 X = -308.2 mm, Y = 326.9 mm, Z = 531.8 mm,       W = -6.7 deg, P = 19.4 deg,
    GP2:
        UF : 1, UT : 2,
       J1 = 0.0 deg, J2 = 0.0 deg
 };
P[134] {
    GP1:
        UF : 6, UT : 5,     CONFIG: 'N U T, 0, 0, 0',
       X = -327.0 mm, Y = 261.3 mm, Z = 531.8 mm,
       W = -6.7 deg, P = 19.5 deg,
    GP2:
        UF : 1, UT : 2,
       J1 = 0.0 deg, J2 = 0.0 deg
 };
P[404] {
    GP1:
        UF : 6, UT : 5,     CONFIG: 'N U T, 0, 0, 0',
 X = -310.0 mm, Y = 332.3 mm, Z = 531.8 mm,       W = -6.7 deg, P = 19.5 deg,
    GP2:
        UF : 1, UT : 2,
       J1 = 0.0 deg, J2 = 0.0 deg
 };
P[135] {
    GP1:
        UF : 6, UT : 5,     CONFIG: 'N U T, 0, 0, 0',
       X = -328.0 mm, Y = 264.4 mm, Z = 531.8 mm,
       W = -7.3 deg, P = 19.2 deg,
    GP2:
        UF : 1, UT : 2,
       J1 = 0.0 deg, J2 = 0.0 deg
 };
P[405] {
    GP1:
        UF : 6, UT : 5,     CONFIG: 'N U T, 0, 0, 0',
 X = -311.0 mm, Y = 335.4 mm, Z = 531.8 mm,       W = -7.3 deg, P = 19.2 deg,
    GP2:
        UF : 1, UT : 2,
       J1 = 0.0 deg, J2 = 0.0 deg
 };
P[136] {
    GP1:
        UF : 6, UT : 5,     CONFIG: 'N U T, 0, 0, 0',
       X = -329.2 mm, Y = 267.4 mm, Z = 531.8 mm,
       W = -7.3 deg, P = 19.0 deg,
    GP2:
        UF : 1, UT : 2,
       J1 = 0.0 deg, J2 = 0.0 deg
 };
P[406] {
    GP1:
        UF : 6, UT : 5,     CONFIG: 'N U T, 0, 0, 0',
 X = -312.2 mm, Y = 338.4 mm, Z = 531.8 mm,       W = -7.3 deg, P = 19.0 deg,
    GP2:
        UF : 1, UT : 2,
       J1 = 0.0 deg, J2 = 0.0 deg
 };
P[137] {
    GP1:
        UF : 6, UT : 5,     CONFIG: 'N U T, 0, 0, 0',
       X = -330.4 mm, Y = 270.7 mm, Z = 531.8 mm,
       W = -7.2 deg, P = 18.9 deg,
    GP2:
        UF : 1, UT : 2,
       J1 = 0.0 deg, J2 = 0.0 deg
 };
P[407] {
    GP1:
        UF : 6, UT : 5,     CONFIG: 'N U T, 0, 0, 0',
 X = -313.4 mm, Y = 341.7 mm, Z = 531.8 mm,       W = -7.2 deg, P = 18.9 deg,
    GP2:
        UF : 1, UT : 2,
       J1 = 0.0 deg, J2 = 0.0 deg
 };
P[138] {
    GP1:
        UF : 6, UT : 5,     CONFIG: 'N U T, 0, 0, 0',
       X = -331.6 mm, Y = 273.8 mm, Z = 531.8 mm,
       W = -7.7 deg, P = 18.5 deg,
    GP2:
        UF : 1, UT : 2,
       J1 = 0.0 deg, J2 = 0.0 deg
 };
P[408] {
    GP1:
        UF : 6, UT : 5,     CONFIG: 'N U T, 0, 0, 0',
 X = -314.6 mm, Y = 344.8 mm, Z = 531.8 mm,       W = -7.7 deg, P = 18.5 deg,
    GP2:
        UF : 1, UT : 2,
       J1 = 0.0 deg, J2 = 0.0 deg
 };
P[139] {
    GP1:
        UF : 6, UT : 5,     CONFIG: 'N U T, 0, 0, 0',
       X = -332.8 mm, Y = 276.8 mm, Z = 531.8 mm,
       W = -7.7 deg, P = 18.5 deg,
    GP2:
        UF : 1, UT : 2,
       J1 = 0.0 deg, J2 = 0.0 deg
 };
P[409] {
    GP1:
        UF : 6, UT : 5,     CONFIG: 'N U T, 0, 0, 0',
 X = -315.8 mm, Y = 347.8 mm, Z = 531.8 mm,       W = -7.7 deg, P = 18.5 deg,
    GP2:
        UF : 1, UT : 2,
       J1 = 0.0 deg, J2 = 0.0 deg
 };
P[140] {
    GP1:
        UF : 6, UT : 5,     CONFIG: 'N U T, 0, 0, 0',
       X = -334.1 mm, Y = 280.0 mm, Z = 531.8 mm,
       W = -7.7 deg, P = 18.4 deg,
    GP2:
        UF : 1, UT : 2,
       J1 = 0.0 deg, J2 = 0.0 deg
 };
P[410] {
    GP1:
        UF : 6, UT : 5,     CONFIG: 'N U T, 0, 0, 0',
 X = -317.1 mm, Y = 351.0 mm, Z = 531.8 mm,       W = -7.7 deg, P = 18.4 deg,
    GP2:
        UF : 1, UT : 2,
       J1 = 0.0 deg, J2 = 0.0 deg
 };
P[141] {
    GP1:
        UF : 6, UT : 5,     CONFIG: 'N U T, 0, 0, 0',
       X = -335.3 mm, Y = 282.9 mm, Z = 531.8 mm,
       W = -8.2 deg, P = 18.1 deg,
    GP2:
        UF : 1, UT : 2,
       J1 = 0.0 deg, J2 = 0.0 deg
 };
P[411] {
    GP1:
        UF : 6, UT : 5,     CONFIG: 'N U T, 0, 0, 0',
 X = -318.3 mm, Y = 353.9 mm, Z = 531.8 mm,       W = -8.2 deg, P = 18.1 deg,
    GP2:
        UF : 1, UT : 2,
       J1 = 0.0 deg, J2 = 0.0 deg
 };
P[142] {
    GP1:
        UF : 6, UT : 5,     CONFIG: 'N U T, 0, 0, 0',
       X = -336.6 mm, Y = 285.8 mm, Z = 531.8 mm,
       W = -8.2 deg, P = 18.0 deg,
    GP2:
        UF : 1, UT : 2,
       J1 = 0.0 deg, J2 = 0.0 deg
 };
P[412] {
    GP1:
        UF : 6, UT : 5,     CONFIG: 'N U T, 0, 0, 0',
 X = -319.6 mm, Y = 356.8 mm, Z = 531.8 mm,       W = -8.2 deg, P = 18.0 deg,
    GP2:
        UF : 1, UT : 2,
       J1 = 0.0 deg, J2 = 0.0 deg
 };
P[143] {
    GP1:
        UF : 6, UT : 5,     CONFIG: 'N U T, 0, 0, 0',
       X = -338.1 mm, Y = 289.2 mm, Z = 531.8 mm,
       W = -8.1 deg, P = 17.9 deg,
    GP2:
        UF : 1, UT : 2,
       J1 = 0.0 deg, J2 = 0.0 deg
 };
P[413] {
    GP1:
        UF : 6, UT : 5,     CONFIG: 'N U T, 0, 0, 0',
 X = -321.1 mm, Y = 360.2 mm, Z = 531.8 mm,       W = -8.1 deg, P = 17.9 deg,
    GP2:
        UF : 1, UT : 2,
       J1 = 0.0 deg, J2 = 0.0 deg
 };
P[144] {
    GP1:
        UF : 6, UT : 5,     CONFIG: 'N U T, 0, 0, 0',
       X = -339.3 mm, Y = 291.9 mm, Z = 531.8 mm,
       W = -8.7 deg, P = 17.5 deg,
    GP2:
        UF : 1, UT : 2,
       J1 = 0.0 deg, J2 = 0.0 deg
 };
P[414] {
    GP1:
        UF : 6, UT : 5,     CONFIG: 'N U T, 0, 0, 0',
 X = -322.3 mm, Y = 362.9 mm, Z = 531.8 mm,       W = -8.7 deg, P = 17.5 deg,
    GP2:
        UF : 1, UT : 2,
       J1 = 0.0 deg, J2 = 0.0 deg
 };
P[145] {
    GP1:
        UF : 6, UT : 5,     CONFIG: 'N U T, 0, 0, 0',
       X = -343.7 mm, Y = 300.7 mm, Z = 531.8 mm,
       W = -9.1 deg, P = 16.9 deg,
    GP2:
        UF : 1, UT : 2,
       J1 = 0.0 deg, J2 = 0.0 deg
 };
P[415] {
    GP1:
        UF : 6, UT : 5,     CONFIG: 'N U T, 0, 0, 0',
 X = -326.7 mm, Y = 371.7 mm, Z = 531.8 mm,       W = -9.1 deg, P = 16.9 deg,
    GP2:
        UF : 1, UT : 2,
       J1 = 0.0 deg, J2 = 0.0 deg
 };
P[146] {
    GP1:
        UF : 6, UT : 5,     CONFIG: 'N U T, 0, 0, 0',
       X = -345.2 mm, Y = 303.6 mm, Z = 531.8 mm,
       W = -9.1 deg, P = 16.8 deg,
    GP2:
        UF : 1, UT : 2,
       J1 = 0.0 deg, J2 = 0.0 deg
 };
P[416] {
    GP1:
        UF : 6, UT : 5,     CONFIG: 'N U T, 0, 0, 0',
 X = -328.2 mm, Y = 374.6 mm, Z = 531.8 mm,       W = -9.1 deg, P = 16.8 deg,
    GP2:
        UF : 1, UT : 2,
       J1 = 0.0 deg, J2 = 0.0 deg
 };
P[147] {
    GP1:
        UF : 6, UT : 5,     CONFIG: 'N U T, 0, 0, 0',
       X = -347.1 mm, Y = 307.0 mm, Z = 531.8 mm,
       W = -9.1 deg, P = 16.7 deg,
    GP2:
        UF : 1, UT : 2,
       J1 = 0.0 deg, J2 = 0.0 deg
 };
P[417] {
    GP1:
        UF : 6, UT : 5,     CONFIG: 'N U T, 0, 0, 0',
 X = -330.1 mm, Y = 378.0 mm, Z = 531.8 mm,       W = -9.1 deg, P = 16.7 deg,
    GP2:
        UF : 1, UT : 2,
       J1 = 0.0 deg, J2 = 0.0 deg
 };
P[148] {
    GP1:
        UF : 6, UT : 5,     CONFIG: 'N U T, 0, 0, 0',
       X = -348.5 mm, Y = 309.7 mm, Z = 531.8 mm,
       W = -9.5 deg, P = 16.4 deg,
    GP2:
        UF : 1, UT : 2,
       J1 = 0.0 deg, J2 = 0.0 deg
 };
P[418] {
    GP1:
        UF : 6, UT : 5,     CONFIG: 'N U T, 0, 0, 0',
 X = -331.5 mm, Y = 380.7 mm, Z = 531.8 mm,       W = -9.5 deg, P = 16.4 deg,
    GP2:
        UF : 1, UT : 2,
       J1 = 0.0 deg, J2 = 0.0 deg
 };
P[149] {
    GP1:
        UF : 6, UT : 5,     CONFIG: 'N U T, 0, 0, 0',
       X = -353.5 mm, Y = 318.3 mm, Z = 531.8 mm,
       W = -9.9 deg, P = 15.9 deg,
    GP2:
        UF : 1, UT : 2,
       J1 = 0.0 deg, J2 = 0.0 deg
 };
P[419] {
    GP1:
        UF : 6, UT : 5,     CONFIG: 'N U T, 0, 0, 0',
 X = -336.5 mm, Y = 389.3 mm, Z = 531.8 mm,       W = -9.9 deg, P = 15.9 deg,
    GP2:
        UF : 1, UT : 2,
       J1 = 0.0 deg, J2 = 0.0 deg
 };
P[150] {
    GP1:
        UF : 6, UT : 5,     CONFIG: 'N U T, 0, 0, 0',
       X = -358.7 mm, Y = 326.6 mm, Z = 531.8 mm,
       W = -10.1 deg, P = 15.4 deg,
    GP2:
        UF : 1, UT : 2,
       J1 = 0.0 deg, J2 = 0.0 deg
 };
P[420] {
    GP1:
        UF : 6, UT : 5,     CONFIG: 'N U T, 0, 0, 0',
 X = -341.7 mm, Y = 397.6 mm, Z = 531.8 mm,       W = -10.1 deg, P = 15.4 deg,
    GP2:
        UF : 1, UT : 2,
       J1 = 0.0 deg, J2 = 0.0 deg
 };
P[151] {
    GP1:
        UF : 6, UT : 5,     CONFIG: 'N U T, 0, 0, 0',
       X = -364.2 mm, Y = 334.9 mm, Z = 531.8 mm,
       W = -10.4 deg, P = 14.9 deg,
    GP2:
        UF : 1, UT : 2,
       J1 = 0.0 deg, J2 = 0.0 deg
 };
P[421] {
    GP1:
        UF : 6, UT : 5,     CONFIG: 'N U T, 0, 0, 0',
 X = -347.2 mm, Y = 405.9 mm, Z = 531.8 mm,       W = -10.4 deg, P = 14.9 deg,
    GP2:
        UF : 1, UT : 2,
       J1 = 0.0 deg, J2 = 0.0 deg
 };
P[152] {
    GP1:
        UF : 6, UT : 5,     CONFIG: 'N U T, 0, 0, 0',
       X = -369.8 mm, Y = 342.9 mm, Z = 531.8 mm,
       W = -10.6 deg, P = 14.5 deg,
    GP2:
        UF : 1, UT : 2,
       J1 = 0.0 deg, J2 = 0.0 deg
 };
P[422] {
    GP1:
        UF : 6, UT : 5,     CONFIG: 'N U T, 0, 0, 0',
 X = -352.8 mm, Y = 413.9 mm, Z = 531.8 mm,       W = -10.6 deg, P = 14.5 deg,
    GP2:
        UF : 1, UT : 2,
       J1 = 0.0 deg, J2 = 0.0 deg
 };
P[153] {
    GP1:
        UF : 6, UT : 5,     CONFIG: 'N U T, 0, 0, 0',
       X = -375.7 mm, Y = 350.9 mm, Z = 531.8 mm,
       W = -11.0 deg, P = 14.1 deg,
    GP2:
        UF : 1, UT : 2,
       J1 = 0.0 deg, J2 = 0.0 deg
 };
P[423] {
    GP1:
        UF : 6, UT : 5,     CONFIG: 'N U T, 0, 0, 0',
 X = -358.7 mm, Y = 421.9 mm, Z = 531.8 mm,       W = -11.0 deg, P = 14.1 deg,
    GP2:
        UF : 1, UT : 2,
       J1 = 0.0 deg, J2 = 0.0 deg
 };
P[154] {
    GP1:
        UF : 6, UT : 5,     CONFIG: 'N U T, 0, 0, 0',
       X = -381.9 mm, Y = 358.6 mm, Z = 531.8 mm,
       W = -11.4 deg, P = 13.8 deg,
    GP2:
        UF : 1, UT : 2,
       J1 = 0.0 deg, J2 = 0.0 deg
 };
P[424] {
    GP1:
        UF : 6, UT : 5,     CONFIG: 'N U T, 0, 0, 0',
 X = -364.9 mm, Y = 429.6 mm, Z = 531.8 mm,       W = -11.4 deg, P = 13.8 deg,
    GP2:
        UF : 1, UT : 2,
       J1 = 0.0 deg, J2 = 0.0 deg
 };
P[155] {
    GP1:
        UF : 6, UT : 5,     CONFIG: 'N U T, 0, 0, 0',
       X = -388.2 mm, Y = 366.1 mm, Z = 531.8 mm,
       W = -11.5 deg, P = 13.2 deg,
    GP2:
        UF : 1, UT : 2,
       J1 = 0.0 deg, J2 = 0.0 deg
 };
P[425] {
    GP1:
        UF : 6, UT : 5,     CONFIG: 'N U T, 0, 0, 0',
 X = -371.2 mm, Y = 437.1 mm, Z = 531.8 mm,       W = -11.5 deg, P = 13.2 deg,
    GP2:
        UF : 1, UT : 2,
       J1 = 0.0 deg, J2 = 0.0 deg
 };
P[156] {
    GP1:
        UF : 6, UT : 5,     CONFIG: 'N U T, 0, 0, 0',
       X = -394.8 mm, Y = 373.5 mm, Z = 531.8 mm,
       W = -11.7 deg, P = 12.5 deg,
    GP2:
        UF : 1, UT : 2,
       J1 = 0.0 deg, J2 = 0.0 deg
 };
P[426] {
    GP1:
        UF : 6, UT : 5,     CONFIG: 'N U T, 0, 0, 0',
 X = -377.8 mm, Y = 444.5 mm, Z = 531.8 mm,       W = -11.7 deg, P = 12.5 deg,
    GP2:
        UF : 1, UT : 2,
       J1 = 0.0 deg, J2 = 0.0 deg
 };
P[157] {
    GP1:
        UF : 6, UT : 5,     CONFIG: 'N U T, 0, 0, 0',
       X = -401.6 mm, Y = 380.6 mm, Z = 531.8 mm,
       W = -11.8 deg, P = 12.0 deg,
    GP2:
        UF : 1, UT : 2,
       J1 = 0.0 deg, J2 = 0.0 deg
 };
P[427] {
    GP1:
        UF : 6, UT : 5,     CONFIG: 'N U T, 0, 0, 0',
 X = -384.6 mm, Y = 451.6 mm, Z = 531.8 mm,       W = -11.8 deg, P = 12.0 deg,
    GP2:
        UF : 1, UT : 2,
       J1 = 0.0 deg, J2 = 0.0 deg
 };
P[158] {
    GP1:
        UF : 6, UT : 5,     CONFIG: 'N U T, 0, 0, 0',
       X = -408.7 mm, Y = 387.5 mm, Z = 531.8 mm,
       W = -11.7 deg, P = 11.3 deg,
    GP2:
        UF : 1, UT : 2,
       J1 = 0.0 deg, J2 = 0.0 deg
 };
P[428] {
    GP1:
        UF : 6, UT : 5,     CONFIG: 'N U T, 0, 0, 0',
 X = -391.7 mm, Y = 458.5 mm, Z = 531.8 mm,       W = -11.7 deg, P = 11.3 deg,
    GP2:
        UF : 1, UT : 2,
       J1 = 0.0 deg, J2 = 0.0 deg
 };
P[159] {
    GP1:
        UF : 6, UT : 5,     CONFIG: 'N U T, 0, 0, 0',
       X = -415.9 mm, Y = 394.3 mm, Z = 531.8 mm,
       W = -11.7 deg, P = 10.7 deg,
    GP2:
        UF : 1, UT : 2,
       J1 = 0.0 deg, J2 = 0.0 deg
 };
P[429] {
    GP1:
        UF : 6, UT : 5,     CONFIG: 'N U T, 0, 0, 0',
 X = -398.9 mm, Y = 465.3 mm, Z = 531.8 mm,       W = -11.7 deg, P = 10.7 deg,
    GP2:
        UF : 1, UT : 2,
       J1 = 0.0 deg, J2 = 0.0 deg
 };
P[160] {
    GP1:
        UF : 6, UT : 5,     CONFIG: 'N U T, 0, 0, 0',
       X = -423.3 mm, Y = 400.8 mm, Z = 531.8 mm,
       W = -11.8 deg, P = 10.1 deg,
    GP2:
        UF : 1, UT : 2,
       J1 = 0.0 deg, J2 = 0.0 deg
 };
P[430] {
    GP1:
        UF : 6, UT : 5,     CONFIG: 'N U T, 0, 0, 0',
 X = -406.3 mm, Y = 471.8 mm, Z = 531.8 mm,       W = -11.8 deg, P = 10.1 deg,
    GP2:
        UF : 1, UT : 2,
       J1 = 0.0 deg, J2 = 0.0 deg
 };
P[161] {
    GP1:
        UF : 6, UT : 5,     CONFIG: 'N U T, 0, 0, 0',
       X = -425.5 mm, Y = 402.6 mm, Z = 531.8 mm,
       W = -11.9 deg, P = 9.9 deg,
    GP2:
        UF : 1, UT : 2,
       J1 = 0.0 deg, J2 = 0.0 deg
 };
P[431] {
    GP1:
        UF : 6, UT : 5,     CONFIG: 'N U T, 0, 0, 0',
 X = -408.5 mm, Y = 473.6 mm, Z = 531.8 mm,       W = -11.9 deg, P = 9.9 deg,
    GP2:
        UF : 1, UT : 2,
       J1 = 0.0 deg, J2 = 0.0 deg
 };
P[162] {
    GP1:
        UF : 6, UT : 5,     CONFIG: 'N U T, 0, 0, 0',
       X = -428.2 mm, Y = 404.9 mm, Z = 531.8 mm,
       W = -11.8 deg, P = 9.8 deg,
    GP2:
        UF : 1, UT : 2,
       J1 = 0.0 deg, J2 = 0.0 deg
 };
P[432] {
    GP1:
        UF : 6, UT : 5,     CONFIG: 'N U T, 0, 0, 0',
 X = -411.2 mm, Y = 475.9 mm, Z = 531.8 mm,       W = -11.8 deg, P = 9.8 deg,
    GP2:
        UF : 1, UT : 2,
       J1 = 0.0 deg, J2 = 0.0 deg
 };
P[163] {
    GP1:
        UF : 6, UT : 5,     CONFIG: 'N U T, 0, 0, 0',
       X = -429.4 mm, Y = 405.9 mm, Z = 531.8 mm,
       W = -11.5 deg, P = 10.1 deg,
    GP2:
        UF : 1, UT : 2,
       J1 = 0.0 deg, J2 = 0.0 deg
 };
P[433] {
    GP1:
        UF : 6, UT : 5,     CONFIG: 'N U T, 0, 0, 0',
 X = -412.4 mm, Y = 476.9 mm, Z = 531.8 mm,       W = -11.5 deg, P = 10.1 deg,
    GP2:
        UF : 1, UT : 2,
       J1 = 0.0 deg, J2 = 0.0 deg
 };
P[164] {
    GP1:
        UF : 6, UT : 5,     CONFIG: 'N U T, 0, 0, 0',
       X = -430.8 mm, Y = 407.1 mm, Z = 531.8 mm,
       W = -11.2 deg, P = 10.8 deg,
    GP2:
        UF : 1, UT : 2,
       J1 = 0.0 deg, J2 = 0.0 deg
 };
P[434] {
    GP1:
        UF : 6, UT : 5,     CONFIG: 'N U T, 0, 0, 0',
 X = -413.8 mm, Y = 478.1 mm, Z = 531.8 mm,       W = -11.2 deg, P = 10.8 deg,
    GP2:
        UF : 1, UT : 2,
       J1 = 0.0 deg, J2 = 0.0 deg
 };
P[165] {
    GP1:
        UF : 6, UT : 5,     CONFIG: 'N U T, 0, 0, 0',
       X = -431.4 mm, Y = 407.7 mm, Z = 531.8 mm,
       W = -11.0 deg, P = 11.1 deg,
    GP2:
        UF : 1, UT : 2,
       J1 = 0.0 deg, J2 = 0.0 deg
 };
P[435] {
    GP1:
        UF : 6, UT : 5,     CONFIG: 'N U T, 0, 0, 0',
 X = -414.4 mm, Y = 478.7 mm, Z = 531.8 mm,       W = -11.0 deg, P = 11.1 deg,
    GP2:
        UF : 1, UT : 2,
       J1 = 0.0 deg, J2 = 0.0 deg
 };
P[166] {
    GP1:
        UF : 6, UT : 5,     CONFIG: 'N U T, 0, 0, 0',
       X = -431.6 mm, Y = 407.9 mm, Z = 531.8 mm,
       W = -10.8 deg, P = 11.3 deg,
    GP2:
        UF : 1, UT : 2,
       J1 = 0.0 deg, J2 = 0.0 deg
 };
P[436] {
    GP1:
        UF : 6, UT : 5,     CONFIG: 'N U T, 0, 0, 0',
 X = -414.6 mm, Y = 478.9 mm, Z = 531.8 mm,       W = -10.8 deg, P = 11.3 deg,
    GP2:
        UF : 1, UT : 2,
       J1 = 0.0 deg, J2 = 0.0 deg
 };
P[167] {
    GP1:
        UF : 6, UT : 5,     CONFIG: 'N U T, 0, 0, 0',
       X = -431.7 mm, Y = 408.1 mm, Z = 531.8 mm,
       W = -10.6 deg, P = 11.6 deg,
    GP2:
        UF : 1, UT : 2,
       J1 = 0.0 deg, J2 = 0.0 deg
 };
P[437] {
    GP1:
        UF : 6, UT : 5,     CONFIG: 'N U T, 0, 0, 0',
 X = -414.7 mm, Y = 479.1 mm, Z = 531.8 mm,       W = -10.6 deg, P = 11.6 deg,
    GP2:
        UF : 1, UT : 2,
       J1 = 0.0 deg, J2 = 0.0 deg
 };
P[168] {
    GP1:
        UF : 6, UT : 5,     CONFIG: 'N U T, 0, 0, 0',
       X = -431.9 mm, Y = 408.2 mm, Z = 531.8 mm,
       W = -10.3 deg, P = 11.8 deg,
    GP2:
        UF : 1, UT : 2,
       J1 = 0.0 deg, J2 = 0.0 deg
 };
P[438] {
    GP1:
        UF : 6, UT : 5,     CONFIG: 'N U T, 0, 0, 0',
 X = -414.9 mm, Y = 479.2 mm, Z = 531.8 mm,       W = -10.3 deg, P = 11.8 deg,
    GP2:
        UF : 1, UT : 2,
       J1 = 0.0 deg, J2 = 0.0 deg
 };
P[169] {
    GP1:
        UF : 6, UT : 5,     CONFIG: 'N U T, 0, 0, 0',
       X = -432.0 mm, Y = 408.4 mm, Z = 531.8 mm,
       W = -10.1 deg, P = 12.1 deg,
    GP2:
        UF : 1, UT : 2,
       J1 = 0.0 deg, J2 = 0.0 deg
 };
P[439] {
    GP1:
        UF : 6, UT : 5,     CONFIG: 'N U T, 0, 0, 0',
 X = -415.0 mm, Y = 479.4 mm, Z = 531.8 mm,       W = -10.1 deg, P = 12.1 deg,
    GP2:
        UF : 1, UT : 2,
       J1 = 0.0 deg, J2 = 0.0 deg
 };
P[170] {
    GP1:
        UF : 6, UT : 5,     CONFIG: 'N U T, 0, 0, 0',
       X = -432.6 mm, Y = 409.1 mm, Z = 531.8 mm,
       W = -9.7 deg, P = 12.7 deg,
    GP2:
        UF : 1, UT : 2,
       J1 = 0.0 deg, J2 = 0.0 deg
 };
P[440] {
    GP1:
        UF : 6, UT : 5,     CONFIG: 'N U T, 0, 0, 0',
 X = -415.6 mm, Y = 480.1 mm, Z = 531.8 mm,       W = -9.7 deg, P = 12.7 deg,
    GP2:
        UF : 1, UT : 2,
       J1 = 0.0 deg, J2 = 0.0 deg
 };
P[171] {
    GP1:
        UF : 6, UT : 5,     CONFIG: 'N U T, 0, 0, 0',
       X = -433.2 mm, Y = 410.0 mm, Z = 531.8 mm,
       W = -9.5 deg, P = 12.9 deg,
    GP2:
        UF : 1, UT : 2,
       J1 = 0.0 deg, J2 = 0.0 deg
 };
P[441] {
    GP1:
        UF : 6, UT : 5,     CONFIG: 'N U T, 0, 0, 0',
 X = -416.2 mm, Y = 481.0 mm, Z = 531.8 mm,       W = -9.5 deg, P = 12.9 deg,
    GP2:
        UF : 1, UT : 2,
       J1 = 0.0 deg, J2 = 0.0 deg
 };
P[172] {
    GP1:
        UF : 6, UT : 5,     CONFIG: 'N U T, 0, 0, 0',
       X = -433.7 mm, Y = 410.7 mm, Z = 531.8 mm,
       W = -8.6 deg, P = 13.4 deg,
    GP2:
        UF : 1, UT : 2,
       J1 = 0.0 deg, J2 = 0.0 deg
 };
P[442] {
    GP1:
        UF : 6, UT : 5,     CONFIG: 'N U T, 0, 0, 0',
 X = -416.7 mm, Y = 481.7 mm, Z = 531.8 mm,       W = -8.6 deg, P = 13.4 deg,
    GP2:
        UF : 1, UT : 2,
       J1 = 0.0 deg, J2 = 0.0 deg
 };
P[173] {
    GP1:
        UF : 6, UT : 5,     CONFIG: 'N U T, 0, 0, 0',
       X = -434.2 mm, Y = 411.5 mm, Z = 531.8 mm,
       W = -7.6 deg, P = 14.0 deg,
    GP2:
        UF : 1, UT : 2,
       J1 = 0.0 deg, J2 = 0.0 deg
 };
P[443] {
    GP1:
        UF : 6, UT : 5,     CONFIG: 'N U T, 0, 0, 0',
 X = -417.2 mm, Y = 482.5 mm, Z = 531.8 mm,       W = -7.6 deg, P = 14.0 deg,
    GP2:
        UF : 1, UT : 2,
       J1 = 0.0 deg, J2 = 0.0 deg
 };
P[174] {
    GP1:
        UF : 6, UT : 5,     CONFIG: 'N U T, 0, 0, 0',
       X = -434.6 mm, Y = 412.3 mm, Z = 531.8 mm,
       W = -7.3 deg, P = 14.0 deg,
    GP2:
        UF : 1, UT : 2,
       J1 = 0.0 deg, J2 = 0.0 deg
 };
P[444] {
    GP1:
        UF : 6, UT : 5,     CONFIG: 'N U T, 0, 0, 0',
 X = -417.6 mm, Y = 483.3 mm, Z = 531.8 mm,       W = -7.3 deg, P = 14.0 deg,
    GP2:
        UF : 1, UT : 2,
       J1 = 0.0 deg, J2 = 0.0 deg
 };
P[175] {
    GP1:
        UF : 6, UT : 5,     CONFIG: 'N U T, 0, 0, 0',
       X = -435.1 mm, Y = 413.3 mm, Z = 531.8 mm,
       W = -6.5 deg, P = 14.3 deg,
    GP2:
        UF : 1, UT : 2,
       J1 = 0.0 deg, J2 = 0.0 deg
 };
P[445] {
    GP1:
        UF : 6, UT : 5,     CONFIG: 'N U T, 0, 0, 0',
 X = -418.1 mm, Y = 484.3 mm, Z = 531.8 mm,       W = -6.5 deg, P = 14.3 deg,
    GP2:
        UF : 1, UT : 2,
       J1 = 0.0 deg, J2 = 0.0 deg
 };
P[176] {
    GP1:
        UF : 6, UT : 5,     CONFIG: 'N U T, 0, 0, 0',
       X = -435.2 mm, Y = 413.6 mm, Z = 531.8 mm,
       W = -6.1 deg, P = 14.4 deg,
    GP2:
        UF : 1, UT : 2,
       J1 = 0.0 deg, J2 = 0.0 deg
 };
P[446] {
    GP1:
        UF : 6, UT : 5,     CONFIG: 'N U T, 0, 0, 0',
 X = -418.2 mm, Y = 484.6 mm, Z = 531.8 mm,       W = -6.1 deg, P = 14.4 deg,
    GP2:
        UF : 1, UT : 2,
       J1 = 0.0 deg, J2 = 0.0 deg
 };
P[177] {
    GP1:
        UF : 6, UT : 5,     CONFIG: 'N U T, 0, 0, 0',
       X = -435.3 mm, Y = 413.8 mm, Z = 531.8 mm,
       W = -5.7 deg, P = 14.5 deg,
    GP2:
        UF : 1, UT : 2,
       J1 = 0.0 deg, J2 = 0.0 deg
 };
P[447] {
    GP1:
        UF : 6, UT : 5,     CONFIG: 'N U T, 0, 0, 0',
 X = -418.3 mm, Y = 484.8 mm, Z = 531.8 mm,       W = -5.7 deg, P = 14.5 deg,
    GP2:
        UF : 1, UT : 2,
       J1 = 0.0 deg, J2 = 0.0 deg
 };
P[178] {
    GP1:
        UF : 6, UT : 5,     CONFIG: 'N U T, 0, 0, 0',
       X = -435.4 mm, Y = 414.1 mm, Z = 531.8 mm,
       W = -5.3 deg, P = 14.5 deg,
    GP2:
        UF : 1, UT : 2,
       J1 = 0.0 deg, J2 = 0.0 deg
 };
P[448] {
    GP1:
        UF : 6, UT : 5,     CONFIG: 'N U T, 0, 0, 0',
 X = -418.4 mm, Y = 485.1 mm, Z = 531.8 mm,       W = -5.3 deg, P = 14.5 deg,
    GP2:
        UF : 1, UT : 2,
       J1 = 0.0 deg, J2 = 0.0 deg
 };
P[179] {
    GP1:
        UF : 6, UT : 5,     CONFIG: 'N U T, 0, 0, 0',
       X = -435.5 mm, Y = 414.3 mm, Z = 531.8 mm,
       W = -5.0 deg, P = 14.6 deg,
    GP2:
        UF : 1, UT : 2,
       J1 = 0.0 deg, J2 = 0.0 deg
 };
P[449] {
    GP1:
        UF : 6, UT : 5,     CONFIG: 'N U T, 0, 0, 0',
 X = -418.5 mm, Y = 485.3 mm, Z = 531.8 mm,       W = -5.0 deg, P = 14.6 deg,
    GP2:
        UF : 1, UT : 2,
       J1 = 0.0 deg, J2 = 0.0 deg
 };
P[180] {
    GP1:
        UF : 6, UT : 5,     CONFIG: 'N U T, 0, 0, 0',
       X = -435.8 mm, Y = 415.4 mm, Z = 531.8 mm,
       W = -4.4 deg, P = 14.5 deg,
    GP2:
        UF : 1, UT : 2,
       J1 = 0.0 deg, J2 = 0.0 deg
 };
P[450] {
    GP1:
        UF : 6, UT : 5,     CONFIG: 'N U T, 0, 0, 0',
 X = -418.8 mm, Y = 486.4 mm, Z = 531.8 mm,       W = -4.4 deg, P = 14.5 deg,
    GP2:
        UF : 1, UT : 2,
       J1 = 0.0 deg, J2 = 0.0 deg
 };
P[181] {
    GP1:
        UF : 6, UT : 5,     CONFIG: 'N U T, 0, 0, 0',
       X = -435.9 mm, Y = 415.7 mm, Z = 531.8 mm,
       W = -4.1 deg, P = 14.4 deg,
    GP2:
        UF : 1, UT : 2,
       J1 = 0.0 deg, J2 = 0.0 deg
 };
P[451] {
    GP1:
        UF : 6, UT : 5,     CONFIG: 'N U T, 0, 0, 0',
 X = -418.9 mm, Y = 486.7 mm, Z = 531.8 mm,       W = -4.1 deg, P = 14.4 deg,
    GP2:
        UF : 1, UT : 2,
       J1 = 0.0 deg, J2 = 0.0 deg
 };
P[182] {
    GP1:
        UF : 6, UT : 5,     CONFIG: 'N U T, 0, 0, 0',
       X = -436.0 mm, Y = 416.0 mm, Z = 531.8 mm,
       W = -3.8 deg, P = 14.4 deg,
    GP2:
        UF : 1, UT : 2,
       J1 = 0.0 deg, J2 = 0.0 deg
 };
P[452] {
    GP1:
        UF : 6, UT : 5,     CONFIG: 'N U T, 0, 0, 0',
 X = -419.0 mm, Y = 487.0 mm, Z = 531.8 mm,       W = -3.8 deg, P = 14.4 deg,
    GP2:
        UF : 1, UT : 2,
       J1 = 0.0 deg, J2 = 0.0 deg
 };
P[183] {
    GP1:
        UF : 6, UT : 5,     CONFIG: 'N U T, 0, 0, 0',
       X = -436.0 mm, Y = 416.2 mm, Z = 531.8 mm,
       W = -3.5 deg, P = 14.4 deg,
    GP2:
        UF : 1, UT : 2,
       J1 = 0.0 deg, J2 = 0.0 deg
 };
P[453] {
    GP1:
        UF : 6, UT : 5,     CONFIG: 'N U T, 0, 0, 0',
 X = -419.0 mm, Y = 487.2 mm, Z = 531.8 mm,       W = -3.5 deg, P = 14.4 deg,
    GP2:
        UF : 1, UT : 2,
       J1 = 0.0 deg, J2 = 0.0 deg
 };
P[184] {
    GP1:
        UF : 6, UT : 5,     CONFIG: 'N U T, 0, 0, 0',
       X = -436.1 mm, Y = 416.5 mm, Z = 531.8 mm,
       W = -3.2 deg, P = 14.4 deg,
    GP2:
        UF : 1, UT : 2,
       J1 = 0.0 deg, J2 = 0.0 deg
 };
P[454] {
    GP1:
        UF : 6, UT : 5,     CONFIG: 'N U T, 0, 0, 0',
 X = -419.1 mm, Y = 487.5 mm, Z = 531.8 mm,       W = -3.2 deg, P = 14.4 deg,
    GP2:
        UF : 1, UT : 2,
       J1 = 0.0 deg, J2 = 0.0 deg
 };
P[185] {
    GP1:
        UF : 6, UT : 5,     CONFIG: 'N U T, 0, 0, 0',
       X = -436.3 mm, Y = 417.8 mm, Z = 531.8 mm,
       W = -2.1 deg, P = 14.2 deg,
    GP2:
        UF : 1, UT : 2,
       J1 = 0.0 deg, J2 = 0.0 deg
 };
P[455] {
    GP1:
        UF : 6, UT : 5,     CONFIG: 'N U T, 0, 0, 0',
 X = -419.3 mm, Y = 488.8 mm, Z = 531.8 mm,       W = -2.1 deg, P = 14.2 deg,
    GP2:
        UF : 1, UT : 2,
       J1 = 0.0 deg, J2 = 0.0 deg
 };
P[186] {
    GP1:
        UF : 6, UT : 5,     CONFIG: 'N U T, 0, 0, 0',
       X = -436.4 mm, Y = 418.6 mm, Z = 531.8 mm,
       W = -1.5 deg, P = 13.9 deg,
    GP2:
        UF : 1, UT : 2,
       J1 = 0.0 deg, J2 = 0.0 deg
 };
P[456] {
    GP1:
        UF : 6, UT : 5,     CONFIG: 'N U T, 0, 0, 0',
 X = -419.4 mm, Y = 489.6 mm, Z = 531.8 mm,       W = -1.5 deg, P = 13.9 deg,
    GP2:
        UF : 1, UT : 2,
       J1 = 0.0 deg, J2 = 0.0 deg
 };
P[187] {
    GP1:
        UF : 6, UT : 5,     CONFIG: 'N U T, 0, 0, 0',
       X = -436.5 mm, Y = 419.0 mm, Z = 531.8 mm,
       W = -1.2 deg, P = 13.8 deg,
    GP2:
        UF : 1, UT : 2,
       J1 = 0.0 deg, J2 = 0.0 deg
 };
P[457] {
    GP1:
        UF : 6, UT : 5,     CONFIG: 'N U T, 0, 0, 0',
 X = -419.5 mm, Y = 490.0 mm, Z = 531.8 mm,       W = -1.2 deg, P = 13.8 deg,
    GP2:
        UF : 1, UT : 2,
       J1 = 0.0 deg, J2 = 0.0 deg
 };
P[188] {
    GP1:
        UF : 6, UT : 5,     CONFIG: 'N U T, 0, 0, 0',
       X = -436.5 mm, Y = 419.4 mm, Z = 531.8 mm,
       W = -1.0 deg, P = 13.6 deg,
    GP2:
        UF : 1, UT : 2,
       J1 = 0.0 deg, J2 = 0.0 deg
 };
P[458] {
    GP1:
        UF : 6, UT : 5,     CONFIG: 'N U T, 0, 0, 0',
 X = -419.5 mm, Y = 490.4 mm, Z = 531.8 mm,       W = -1.0 deg, P = 13.6 deg,
    GP2:
        UF : 1, UT : 2,
       J1 = 0.0 deg, J2 = 0.0 deg
 };
P[189] {
    GP1:
        UF : 6, UT : 5,     CONFIG: 'N U T, 0, 0, 0',
       X = -436.5 mm, Y = 419.8 mm, Z = 531.8 mm,
       W = -0.6 deg, P = 13.4 deg,
    GP2:
        UF : 1, UT : 2,
       J1 = 0.0 deg, J2 = 0.0 deg
 };
P[459] {
    GP1:
        UF : 6, UT : 5,     CONFIG: 'N U T, 0, 0, 0',
 X = -419.5 mm, Y = 490.8 mm, Z = 531.8 mm,       W = -0.6 deg, P = 13.4 deg,
    GP2:
        UF : 1, UT : 2,
       J1 = 0.0 deg, J2 = 0.0 deg
 };
P[190] {
    GP1:
        UF : 6, UT : 5,     CONFIG: 'N U T, 0, 0, 0',
       X = -436.5 mm, Y = 420.2 mm, Z = 531.8 mm,
       W = -0.4 deg, P = 13.2 deg,
    GP2:
        UF : 1, UT : 2,
       J1 = 0.0 deg, J2 = 0.0 deg
 };
P[460] {
    GP1:
        UF : 6, UT : 5,     CONFIG: 'N U T, 0, 0, 0',
 X = -419.5 mm, Y = 491.2 mm, Z = 531.8 mm,       W = -0.4 deg, P = 13.2 deg,
    GP2:
        UF : 1, UT : 2,
       J1 = 0.0 deg, J2 = 0.0 deg
 };
P[191] {
    GP1:
        UF : 6, UT : 5,     CONFIG: 'N U T, 0, 0, 0',
       X = -436.5 mm, Y = 420.5 mm, Z = 531.8 mm,
       W = 0.0 deg, P = 13.0 deg,
    GP2:
        UF : 1, UT : 2,
       J1 = 0.0 deg, J2 = 0.0 deg
 };
P[461] {
    GP1:
        UF : 6, UT : 5,     CONFIG: 'N U T, 0, 0, 0',
 X = -419.5 mm, Y = 491.5 mm, Z = 531.8 mm,       W = 0.0 deg, P = 13.0 deg,
    GP2:
        UF : 1, UT : 2,
       J1 = 0.0 deg, J2 = 0.0 deg
 };
P[192] {
    GP1:
        UF : 6, UT : 5,     CONFIG: 'N U T, 0, 0, 0',
       X = -436.6 mm, Y = 420.9 mm, Z = 531.8 mm,
       W = 0.3 deg, P = 12.8 deg,
    GP2:
        UF : 1, UT : 2,
       J1 = 0.0 deg, J2 = 0.0 deg
 };
P[462] {
    GP1:
        UF : 6, UT : 5,     CONFIG: 'N U T, 0, 0, 0',
 X = -419.6 mm, Y = 491.9 mm, Z = 531.8 mm,       W = 0.3 deg, P = 12.8 deg,
    GP2:
        UF : 1, UT : 2,
       J1 = 0.0 deg, J2 = 0.0 deg
 };
P[193] {
    GP1:
        UF : 6, UT : 5,     CONFIG: 'N U T, 0, 0, 0',
       X = -436.5 mm, Y = 422.0 mm, Z = 531.8 mm,
       W = 0.7 deg, P = 12.6 deg,
    GP2:
        UF : 1, UT : 2,
       J1 = 0.0 deg, J2 = 0.0 deg
 };
P[463] {
    GP1:
        UF : 6, UT : 5,     CONFIG: 'N U T, 0, 0, 0',
 X = -419.5 mm, Y = 493.0 mm, Z = 531.8 mm,       W = 0.7 deg, P = 12.6 deg,
    GP2:
        UF : 1, UT : 2,
       J1 = 0.0 deg, J2 = 0.0 deg
 };
P[194] {
    GP1:
        UF : 6, UT : 5,     CONFIG: 'N U T, 0, 0, 0',
       X = -436.5 mm, Y = 422.2 mm, Z = 531.8 mm,
       W = 0.9 deg, P = 12.5 deg,
    GP2:
        UF : 1, UT : 2,
       J1 = 0.0 deg, J2 = 0.0 deg
 };
P[464] {
    GP1:
        UF : 6, UT : 5,     CONFIG: 'N U T, 0, 0, 0',
 X = -419.5 mm, Y = 493.2 mm, Z = 531.8 mm,       W = 0.9 deg, P = 12.5 deg,
    GP2:
        UF : 1, UT : 2,
       J1 = 0.0 deg, J2 = 0.0 deg
 };
P[195] {
    GP1:
        UF : 6, UT : 5,     CONFIG: 'N U T, 0, 0, 0',
       X = -436.5 mm, Y = 422.4 mm, Z = 531.8 mm,
       W = 1.2 deg, P = 12.5 deg,
    GP2:
        UF : 1, UT : 2,
       J1 = 0.0 deg, J2 = 0.0 deg
 };
P[465] {
    GP1:
        UF : 6, UT : 5,     CONFIG: 'N U T, 0, 0, 0',
 X = -419.5 mm, Y = 493.4 mm, Z = 531.8 mm,       W = 1.2 deg, P = 12.5 deg,
    GP2:
        UF : 1, UT : 2,
       J1 = 0.0 deg, J2 = 0.0 deg
 };
P[196] {
    GP1:
        UF : 6, UT : 5,     CONFIG: 'N U T, 0, 0, 0',
       X = -436.5 mm, Y = 422.5 mm, Z = 531.8 mm,
       W = 1.4 deg, P = 12.4 deg,
    GP2:
        UF : 1, UT : 2,
       J1 = 0.0 deg, J2 = 0.0 deg
 };
P[466] {
    GP1:
        UF : 6, UT : 5,     CONFIG: 'N U T, 0, 0, 0',
 X = -419.5 mm, Y = 493.5 mm, Z = 531.8 mm,       W = 1.4 deg, P = 12.4 deg,
    GP2:
        UF : 1, UT : 2,
       J1 = 0.0 deg, J2 = 0.0 deg
 };
P[197] {
    GP1:
        UF : 6, UT : 5,     CONFIG: 'N U T, 0, 0, 0',
       X = -436.5 mm, Y = 422.7 mm, Z = 531.8 mm,
       W = 1.6 deg, P = 12.3 deg,
    GP2:
        UF : 1, UT : 2,
       J1 = 0.0 deg, J2 = 0.0 deg
 };
P[467] {
    GP1:
        UF : 6, UT : 5,     CONFIG: 'N U T, 0, 0, 0',
 X = -419.5 mm, Y = 493.7 mm, Z = 531.8 mm,       W = 1.6 deg, P = 12.3 deg,
    GP2:
        UF : 1, UT : 2,
       J1 = 0.0 deg, J2 = 0.0 deg
 };
P[198] {
    GP1:
        UF : 6, UT : 5,     CONFIG: 'N U T, 0, 0, 0',
       X = -436.4 mm, Y = 423.4 mm, Z = 531.8 mm,
       W = 2.2 deg, P = 11.6 deg,
    GP2:
        UF : 1, UT : 2,
       J1 = 0.0 deg, J2 = 0.0 deg
 };
P[468] {
    GP1:
        UF : 6, UT : 5,     CONFIG: 'N U T, 0, 0, 0',
 X = -419.4 mm, Y = 494.4 mm, Z = 531.8 mm,       W = 2.2 deg, P = 11.6 deg,
    GP2:
        UF : 1, UT : 2,
       J1 = 0.0 deg, J2 = 0.0 deg
 };
P[199] {
    GP1:
        UF : 6, UT : 5,     CONFIG: 'N U T, 0, 0, 0',
       X = -436.2 mm, Y = 424.2 mm, Z = 531.8 mm,
       W = 2.3 deg, P = 11.1 deg,
    GP2:
        UF : 1, UT : 2,
       J1 = 0.0 deg, J2 = 0.0 deg
 };
P[469] {
    GP1:
        UF : 6, UT : 5,     CONFIG: 'N U T, 0, 0, 0',
 X = -419.2 mm, Y = 495.2 mm, Z = 531.8 mm,       W = 2.3 deg, P = 11.1 deg,
    GP2:
        UF : 1, UT : 2,
       J1 = 0.0 deg, J2 = 0.0 deg
 };
P[200] {
    GP1:
        UF : 6, UT : 5,     CONFIG: 'N U T, 0, 0, 0',
       X = -436.0 mm, Y = 425.1 mm, Z = 531.8 mm,
       W = 2.6 deg, P = 11.0 deg,
    GP2:
        UF : 1, UT : 2,
       J1 = 0.0 deg, J2 = 0.0 deg
 };
P[470] {
    GP1:
        UF : 6, UT : 5,     CONFIG: 'N U T, 0, 0, 0',
 X = -419.0 mm, Y = 496.1 mm, Z = 531.8 mm,       W = 2.6 deg, P = 11.0 deg,
    GP2:
        UF : 1, UT : 2,
       J1 = 0.0 deg, J2 = 0.0 deg
 };
P[201] {
    GP1:
        UF : 6, UT : 5,     CONFIG: 'N U T, 0, 0, 0',
       X = -435.9 mm, Y = 425.4 mm, Z = 531.8 mm,
       W = 2.7 deg, P = 10.6 deg,
    GP2:
        UF : 1, UT : 2,
       J1 = 0.0 deg, J2 = 0.0 deg
 };
P[471] {
    GP1:
        UF : 6, UT : 5,     CONFIG: 'N U T, 0, 0, 0',
 X = -418.9 mm, Y = 496.4 mm, Z = 531.8 mm,       W = 2.7 deg, P = 10.6 deg,
    GP2:
        UF : 1, UT : 2,
       J1 = 0.0 deg, J2 = 0.0 deg
 };
P[202] {
    GP1:
        UF : 6, UT : 5,     CONFIG: 'N U T, 0, 0, 0',
       X = -435.9 mm, Y = 425.7 mm, Z = 531.8 mm,
       W = 2.9 deg, P = 10.2 deg,
    GP2:
        UF : 1, UT : 2,
       J1 = 0.0 deg, J2 = 0.0 deg
 };
P[472] {
    GP1:
        UF : 6, UT : 5,     CONFIG: 'N U T, 0, 0, 0',
 X = -418.9 mm, Y = 496.7 mm, Z = 531.8 mm,       W = 2.9 deg, P = 10.2 deg,
    GP2:
        UF : 1, UT : 2,
       J1 = 0.0 deg, J2 = 0.0 deg
 };
P[203] {
    GP1:
        UF : 6, UT : 5,     CONFIG: 'N U T, 0, 0, 0',
       X = -435.8 mm, Y = 425.9 mm, Z = 531.8 mm,
       W = 3.0 deg, P = 9.8 deg,
    GP2:
        UF : 1, UT : 2,
       J1 = 0.0 deg, J2 = 0.0 deg
 };
P[473] {
    GP1:
        UF : 6, UT : 5,     CONFIG: 'N U T, 0, 0, 0',
 X = -418.8 mm, Y = 496.9 mm, Z = 531.8 mm,       W = 3.0 deg, P = 9.8 deg,
    GP2:
        UF : 1, UT : 2,
       J1 = 0.0 deg, J2 = 0.0 deg
 };
P[204] {
    GP1:
        UF : 6, UT : 5,     CONFIG: 'N U T, 0, 0, 0',
       X = -435.7 mm, Y = 426.2 mm, Z = 531.8 mm,
       W = 3.2 deg, P = 9.4 deg,
    GP2:
        UF : 1, UT : 2,
       J1 = 0.0 deg, J2 = 0.0 deg
 };
P[474] {
    GP1:
        UF : 6, UT : 5,     CONFIG: 'N U T, 0, 0, 0',
 X = -418.7 mm, Y = 497.2 mm, Z = 531.8 mm,       W = 3.2 deg, P = 9.4 deg,
    GP2:
        UF : 1, UT : 2,
       J1 = 0.0 deg, J2 = 0.0 deg
 };
P[205] {
    GP1:
        UF : 6, UT : 5,     CONFIG: 'N U T, 0, 0, 0',
       X = -435.3 mm, Y = 427.3 mm, Z = 531.8 mm,
       W = 3.4 deg, P = 8.6 deg,
    GP2:
        UF : 1, UT : 2,
       J1 = 0.0 deg, J2 = 0.0 deg
 };
P[475] {
    GP1:
        UF : 6, UT : 5,     CONFIG: 'N U T, 0, 0, 0',
 X = -418.3 mm, Y = 498.3 mm, Z = 531.8 mm,       W = 3.4 deg, P = 8.6 deg,
    GP2:
        UF : 1, UT : 2,
       J1 = 0.0 deg, J2 = 0.0 deg
 };
P[206] {
    GP1:
        UF : 6, UT : 5,     CONFIG: 'N U T, 0, 0, 0',
       X = -434.9 mm, Y = 428.2 mm, Z = 531.8 mm,
       W = 3.4 deg, P = 7.5 deg,
    GP2:
        UF : 1, UT : 2,
       J1 = 0.0 deg, J2 = 0.0 deg
 };
P[476] {
    GP1:
        UF : 6, UT : 5,     CONFIG: 'N U T, 0, 0, 0',
 X = -417.9 mm, Y = 499.2 mm, Z = 531.8 mm,       W = 3.4 deg, P = 7.5 deg,
    GP2:
        UF : 1, UT : 2,
       J1 = 0.0 deg, J2 = 0.0 deg
 };
P[207] {
    GP1:
        UF : 6, UT : 5,     CONFIG: 'N U T, 0, 0, 0',
       X = -434.8 mm, Y = 428.4 mm, Z = 531.8 mm,
       W = 3.4 deg, P = 7.3 deg,
    GP2:
        UF : 1, UT : 2,
       J1 = 0.0 deg, J2 = 0.0 deg
 };
P[477] {
    GP1:
        UF : 6, UT : 5,     CONFIG: 'N U T, 0, 0, 0',
 X = -417.8 mm, Y = 499.4 mm, Z = 531.8 mm,       W = 3.4 deg, P = 7.3 deg,
    GP2:
        UF : 1, UT : 2,
       J1 = 0.0 deg, J2 = 0.0 deg
 };
P[208] {
    GP1:
        UF : 6, UT : 5,     CONFIG: 'N U T, 0, 0, 0',
       X = -434.7 mm, Y = 428.7 mm, Z = 531.8 mm,
       W = 3.5 deg, P = 7.0 deg,
    GP2:
        UF : 1, UT : 2,
       J1 = 0.0 deg, J2 = 0.0 deg
 };
P[478] {
    GP1:
        UF : 6, UT : 5,     CONFIG: 'N U T, 0, 0, 0',
 X = -417.7 mm, Y = 499.7 mm, Z = 531.8 mm,       W = 3.5 deg, P = 7.0 deg,
    GP2:
        UF : 1, UT : 2,
       J1 = 0.0 deg, J2 = 0.0 deg
 };
P[209] {
    GP1:
        UF : 6, UT : 5,     CONFIG: 'N U T, 0, 0, 0',
       X = -434.6 mm, Y = 428.9 mm, Z = 531.8 mm,
       W = 3.5 deg, P = 6.7 deg,
    GP2:
        UF : 1, UT : 2,
       J1 = 0.0 deg, J2 = 0.0 deg
 };
P[479] {
    GP1:
        UF : 6, UT : 5,     CONFIG: 'N U T, 0, 0, 0',
 X = -417.6 mm, Y = 499.9 mm, Z = 531.8 mm,       W = 3.5 deg, P = 6.7 deg,
    GP2:
        UF : 1, UT : 2,
       J1 = 0.0 deg, J2 = 0.0 deg
 };
P[210] {
    GP1:
        UF : 6, UT : 5,     CONFIG: 'N U T, 0, 0, 0',
       X = -434.5 mm, Y = 429.1 mm, Z = 531.8 mm,
       W = 3.5 deg, P = 6.4 deg,
    GP2:
        UF : 1, UT : 2,
       J1 = 0.0 deg, J2 = 0.0 deg
 };
P[480] {
    GP1:
        UF : 6, UT : 5,     CONFIG: 'N U T, 0, 0, 0',
 X = -417.5 mm, Y = 500.1 mm, Z = 531.8 mm,       W = 3.5 deg, P = 6.4 deg,
    GP2:
        UF : 1, UT : 2,
       J1 = 0.0 deg, J2 = 0.0 deg
 };
P[211] {
    GP1:
        UF : 6, UT : 5,     CONFIG: 'N U T, 0, 0, 0',
       X = -434.0 mm, Y = 429.9 mm, Z = 531.8 mm,
       W = 3.4 deg, P = 5.8 deg,
    GP2:
        UF : 1, UT : 2,
       J1 = 0.0 deg, J2 = 0.0 deg
 };
P[481] {
    GP1:
        UF : 6, UT : 5,     CONFIG: 'N U T, 0, 0, 0',
 X = -417.0 mm, Y = 500.9 mm, Z = 531.8 mm,       W = 3.4 deg, P = 5.8 deg,
    GP2:
        UF : 1, UT : 2,
       J1 = 0.0 deg, J2 = 0.0 deg
 };
P[212] {
    GP1:
        UF : 6, UT : 5,     CONFIG: 'N U T, 0, 0, 0',
       X = -433.8 mm, Y = 430.3 mm, Z = 531.8 mm,
       W = 3.4 deg, P = 5.5 deg,
    GP2:
        UF : 1, UT : 2,
       J1 = 0.0 deg, J2 = 0.0 deg
 };
P[482] {
    GP1:
        UF : 6, UT : 5,     CONFIG: 'N U T, 0, 0, 0',
 X = -416.8 mm, Y = 501.3 mm, Z = 531.8 mm,       W = 3.4 deg, P = 5.5 deg,
    GP2:
        UF : 1, UT : 2,
       J1 = 0.0 deg, J2 = 0.0 deg
 };
P[213] {
    GP1:
        UF : 6, UT : 5,     CONFIG: 'N U T, 0, 0, 0',
       X = -433.5 mm, Y = 430.7 mm, Z = 531.8 mm,
       W = 3.3 deg, P = 5.2 deg,
    GP2:
        UF : 1, UT : 2,
       J1 = 0.0 deg, J2 = 0.0 deg
 };
P[483] {
    GP1:
        UF : 6, UT : 5,     CONFIG: 'N U T, 0, 0, 0',
 X = -416.5 mm, Y = 501.7 mm, Z = 531.8 mm,       W = 3.3 deg, P = 5.2 deg,
    GP2:
        UF : 1, UT : 2,
       J1 = 0.0 deg, J2 = 0.0 deg
 };
P[214] {
    GP1:
        UF : 6, UT : 5,     CONFIG: 'N U T, 0, 0, 0',
       X = -433.2 mm, Y = 431.1 mm, Z = 531.8 mm,
       W = 3.3 deg, P = 4.8 deg,
    GP2:
        UF : 1, UT : 2,
       J1 = 0.0 deg, J2 = 0.0 deg
 };
P[484] {
    GP1:
        UF : 6, UT : 5,     CONFIG: 'N U T, 0, 0, 0',
 X = -416.2 mm, Y = 502.1 mm, Z = 531.8 mm,       W = 3.3 deg, P = 4.8 deg,
    GP2:
        UF : 1, UT : 2,
       J1 = 0.0 deg, J2 = 0.0 deg
 };
P[215] {
    GP1:
        UF : 6, UT : 5,     CONFIG: 'N U T, 0, 0, 0',
       X = -433.0 mm, Y = 431.5 mm, Z = 531.8 mm,
       W = 3.2 deg, P = 4.5 deg,
    GP2:
        UF : 1, UT : 2,
       J1 = 0.0 deg, J2 = 0.0 deg
 };
P[485] {
    GP1:
        UF : 6, UT : 5,     CONFIG: 'N U T, 0, 0, 0',
 X = -416.0 mm, Y = 502.5 mm, Z = 531.8 mm,       W = 3.2 deg, P = 4.5 deg,
    GP2:
        UF : 1, UT : 2,
       J1 = 0.0 deg, J2 = 0.0 deg
 };
P[216] {
    GP1:
        UF : 6, UT : 5,     CONFIG: 'N U T, 0, 0, 0',
       X = -432.7 mm, Y = 431.9 mm, Z = 531.8 mm,
       W = 3.2 deg, P = 4.2 deg,
    GP2:
        UF : 1, UT : 2,
       J1 = 0.0 deg, J2 = 0.0 deg
 };
P[486] {
    GP1:
        UF : 6, UT : 5,     CONFIG: 'N U T, 0, 0, 0',
 X = -415.7 mm, Y = 502.9 mm, Z = 531.8 mm,       W = 3.2 deg, P = 4.2 deg,
    GP2:
        UF : 1, UT : 2,
       J1 = 0.0 deg, J2 = 0.0 deg
 };
P[217] {
    GP1:
        UF : 6, UT : 5,     CONFIG: 'N U T, 0, 0, 0',
       X = -432.4 mm, Y = 432.3 mm, Z = 531.8 mm,
       W = 3.0 deg, P = 3.9 deg,
    GP2:
        UF : 1, UT : 2,
       J1 = 0.0 deg, J2 = 0.0 deg
 };
P[487] {
    GP1:
        UF : 6, UT : 5,     CONFIG: 'N U T, 0, 0, 0',
 X = -415.4 mm, Y = 503.3 mm, Z = 531.8 mm,       W = 3.0 deg, P = 3.9 deg,
    GP2:
        UF : 1, UT : 2,
       J1 = 0.0 deg, J2 = 0.0 deg
 };
P[218] {
    GP1:
        UF : 6, UT : 5,     CONFIG: 'N U T, 0, 0, 0',
       X = -431.6 mm, Y = 433.2 mm, Z = 531.8 mm,
       W = 3.2 deg, P = 3.7 deg,
    GP2:
        UF : 1, UT : 2,
       J1 = 0.0 deg, J2 = 0.0 deg
 };
P[488] {
    GP1:
        UF : 6, UT : 5,     CONFIG: 'N U T, 0, 0, 0',
 X = -414.6 mm, Y = 504.2 mm, Z = 531.8 mm,       W = 3.2 deg, P = 3.7 deg,
    GP2:
        UF : 1, UT : 2,
       J1 = 0.0 deg, J2 = 0.0 deg
 };
P[219] {
    GP1:
        UF : 6, UT : 5,     CONFIG: 'N U T, 0, 0, 0',
       X = -430.8 mm, Y = 434.1 mm, Z = 531.8 mm,
       W = 3.2 deg, P = 3.4 deg,
    GP2:
        UF : 1, UT : 2,
       J1 = 0.0 deg, J2 = 0.0 deg
 };
P[489] {
    GP1:
        UF : 6, UT : 5,     CONFIG: 'N U T, 0, 0, 0',
 X = -413.8 mm, Y = 505.1 mm, Z = 531.8 mm,       W = 3.2 deg, P = 3.4 deg,
    GP2:
        UF : 1, UT : 2,
       J1 = 0.0 deg, J2 = 0.0 deg
 };
P[220] {
    GP1:
        UF : 6, UT : 5,     CONFIG: 'N U T, 0, 0, 0',
       X = -424.1 mm, Y = 441.2 mm, Z = 531.8 mm,
       W = 2.8 deg, P = 3.0 deg,
    GP2:
        UF : 1, UT : 2,
       J1 = 0.0 deg, J2 = 0.0 deg
 };
P[490] {
    GP1:
        UF : 6, UT : 5,     CONFIG: 'N U T, 0, 0, 0',
 X = -407.1 mm, Y = 512.2 mm, Z = 531.8 mm,       W = 2.8 deg, P = 3.0 deg,
    GP2:
        UF : 1, UT : 2,
       J1 = 0.0 deg, J2 = 0.0 deg
 };
P[221] {
    GP1:
        UF : 6, UT : 5,     CONFIG: 'N U T, 0, 0, 0',
       X = -417.2 mm, Y = 448.3 mm, Z = 531.8 mm,
       W = 2.4 deg, P = 2.6 deg,
    GP2:
        UF : 1, UT : 2,
       J1 = 0.0 deg, J2 = 0.0 deg
 };
P[491] {
    GP1:
        UF : 6, UT : 5,     CONFIG: 'N U T, 0, 0, 0',
 X = -400.2 mm, Y = 519.3 mm, Z = 531.8 mm,       W = 2.4 deg, P = 2.6 deg,
    GP2:
        UF : 1, UT : 2,
       J1 = 0.0 deg, J2 = 0.0 deg
 };
P[222] {
    GP1:
        UF : 6, UT : 5,     CONFIG: 'N U T, 0, 0, 0',
       X = -410.4 mm, Y = 455.4 mm, Z = 531.8 mm,
       W = 2.1 deg, P = 2.2 deg,
    GP2:
        UF : 1, UT : 2,
       J1 = 0.0 deg, J2 = 0.0 deg
 };
P[492] {
    GP1:
        UF : 6, UT : 5,     CONFIG: 'N U T, 0, 0, 0',
 X = -393.4 mm, Y = 526.4 mm, Z = 531.8 mm,       W = 2.1 deg, P = 2.2 deg,
    GP2:
        UF : 1, UT : 2,
       J1 = 0.0 deg, J2 = 0.0 deg
 };
P[223] {
    GP1:
        UF : 6, UT : 5,     CONFIG: 'N U T, 0, 0, 0',
       X = -403.4 mm, Y = 462.4 mm, Z = 531.8 mm,
       W = 1.7 deg, P = 1.8 deg,
    GP2:
        UF : 1, UT : 2,
       J1 = 0.0 deg, J2 = 0.0 deg
 };
P[493] {
    GP1:
        UF : 6, UT : 5,     CONFIG: 'N U T, 0, 0, 0',
 X = -386.4 mm, Y = 533.4 mm, Z = 531.8 mm,       W = 1.7 deg, P = 1.8 deg,
    GP2:
        UF : 1, UT : 2,
       J1 = 0.0 deg, J2 = 0.0 deg
 };
P[224] {
    GP1:
        UF : 6, UT : 5,     CONFIG: 'N U T, 0, 0, 0',
       X = -399.0 mm, Y = 466.8 mm, Z = 531.8 mm,
       W = 1.5 deg, P = 1.6 deg,
    GP2:
        UF : 1, UT : 2,
       J1 = 0.0 deg, J2 = 0.0 deg
 };
P[494] {
    GP1:
        UF : 6, UT : 5,     CONFIG: 'N U T, 0, 0, 0',
 X = -382.0 mm, Y = 537.8 mm, Z = 531.8 mm,       W = 1.5 deg, P = 1.6 deg,
    GP2:
        UF : 1, UT : 2,
       J1 = 0.0 deg, J2 = 0.0 deg
 };
P[225] {
    GP1:
        UF : 6, UT : 5,     CONFIG: 'N U T, 0, 0, 0',
       X = -392.0 mm, Y = 473.2 mm, Z = 531.8 mm,
       W = 1.1 deg, P = 1.2 deg,
    GP2:
        UF : 1, UT : 2,
       J1 = 0.0 deg, J2 = 0.0 deg
 };
P[495] {
    GP1:
        UF : 6, UT : 5,     CONFIG: 'N U T, 0, 0, 0',
 X = -375.0 mm, Y = 544.2 mm, Z = 531.8 mm,       W = 1.1 deg, P = 1.2 deg,
    GP2:
        UF : 1, UT : 2,
       J1 = 0.0 deg, J2 = 0.0 deg
 };
P[226] {
    GP1:
        UF : 6, UT : 5,     CONFIG: 'N U T, 0, 0, 0',
       X = -384.7 mm, Y = 479.5 mm, Z = 531.8 mm,
       W = 0.8 deg, P = 0.9 deg,
    GP2:
        UF : 1, UT : 2,
       J1 = 0.0 deg, J2 = 0.0 deg
 };
P[496] {
    GP1:
        UF : 6, UT : 5,     CONFIG: 'N U T, 0, 0, 0',
 X = -367.7 mm, Y = 550.5 mm, Z = 531.8 mm,       W = 0.8 deg, P = 0.9 deg,
    GP2:
        UF : 1, UT : 2,
       J1 = 0.0 deg, J2 = 0.0 deg
 };
P[227] {
    GP1:
        UF : 6, UT : 5,     CONFIG: 'N U T, 0, 0, 0',
       X = -383.4 mm, Y = 481.0 mm, Z = 531.8 mm,
       W = 0.7 deg, P = 0.7 deg,
    GP2:
        UF : 1, UT : 2,
       J1 = 0.0 deg, J2 = 0.0 deg
 };
P[497] {
    GP1:
        UF : 6, UT : 5,     CONFIG: 'N U T, 0, 0, 0',
 X = -366.4 mm, Y = 552.0 mm, Z = 531.8 mm,       W = 0.7 deg, P = 0.7 deg,
    GP2:
        UF : 1, UT : 2,
       J1 = 0.0 deg, J2 = 0.0 deg
 };
P[228] {
    GP1:
        UF : 6, UT : 5,     CONFIG: 'N U T, 0, 0, 0',
       X = -382.6 mm, Y = 482.2 mm, Z = 531.8 mm,
       W = 0.7 deg, P = 0.7 deg,
    GP2:
        UF : 1, UT : 2,
       J1 = 0.0 deg, J2 = 0.0 deg
 };
P[498] {
    GP1:
        UF : 6, UT : 5,     CONFIG: 'N U T, 0, 0, 0',
 X = -365.6 mm, Y = 553.2 mm, Z = 531.8 mm,       W = 0.7 deg, P = 0.7 deg,
    GP2:
        UF : 1, UT : 2,
       J1 = 0.0 deg, J2 = 0.0 deg
 };
P[229] {
    GP1:
        UF : 6, UT : 5,     CONFIG: 'N U T, 0, 0, 0',
       X = -382.0 mm, Y = 483.3 mm, Z = 531.8 mm,
       W = 0.6 deg, P = 0.7 deg,
    GP2:
        UF : 1, UT : 2,
       J1 = 0.0 deg, J2 = 0.0 deg
 };
P[499] {
    GP1:
        UF : 6, UT : 5,     CONFIG: 'N U T, 0, 0, 0',
 X = -365.0 mm, Y = 554.3 mm, Z = 531.8 mm,       W = 0.6 deg, P = 0.7 deg,
    GP2:
        UF : 1, UT : 2,
       J1 = 0.0 deg, J2 = 0.0 deg
 };
P[230] {
    GP1:
        UF : 6, UT : 5,     CONFIG: 'N U T, 0, 0, 0',
       X = -381.7 mm, Y = 484.2 mm, Z = 531.8 mm,
       W = 0.6 deg, P = 0.6 deg,
    GP2:
        UF : 1, UT : 2,
       J1 = 0.0 deg, J2 = 0.0 deg
 };
P[500] {
    GP1:
        UF : 6, UT : 5,     CONFIG: 'N U T, 0, 0, 0',
 X = -364.7 mm, Y = 555.2 mm, Z = 531.8 mm,       W = 0.6 deg, P = 0.6 deg,
    GP2:
        UF : 1, UT : 2,
       J1 = 0.0 deg, J2 = 0.0 deg
 };
P[231] {
    GP1:
        UF : 6, UT : 5,     CONFIG: 'N U T, 0, 0, 0',
       X = -381.3 mm, Y = 485.3 mm, Z = 531.8 mm,
       W = 0.5 deg, P = 0.6 deg,
    GP2:
        UF : 1, UT : 2,
       J1 = 0.0 deg, J2 = 0.0 deg
 };
P[501] {
    GP1:
        UF : 6, UT : 5,     CONFIG: 'N U T, 0, 0, 0',
 X = -364.3 mm, Y = 556.3 mm, Z = 531.8 mm,       W = 0.5 deg, P = 0.6 deg,
    GP2:
        UF : 1, UT : 2,
       J1 = 0.0 deg, J2 = 0.0 deg
 };
P[232] {
    GP1:
        UF : 6, UT : 5,     CONFIG: 'N U T, 0, 0, 0',
       X = -381.0 mm, Y = 486.6 mm, Z = 531.8 mm,
       W = 0.5 deg, P = 0.5 deg,
    GP2:
        UF : 1, UT : 2,
       J1 = 0.0 deg, J2 = 0.0 deg
 };
P[502] {
    GP1:
        UF : 6, UT : 5,     CONFIG: 'N U T, 0, 0, 0',
 X = -364.0 mm, Y = 557.6 mm, Z = 531.8 mm,       W = 0.5 deg, P = 0.5 deg,
    GP2:
        UF : 1, UT : 2,
       J1 = 0.0 deg, J2 = 0.0 deg
 };
P[233] {
    GP1:
        UF : 6, UT : 5,     CONFIG: 'N U T, 0, 0, 0',
       X = -380.9 mm, Y = 488.8 mm, Z = 531.8 mm,
       W = 0.4 deg, P = 0.5 deg,
    GP2:
        UF : 1, UT : 2,
       J1 = 0.0 deg, J2 = 0.0 deg
 };
P[503] {
    GP1:
        UF : 6, UT : 5,     CONFIG: 'N U T, 0, 0, 0',
 X = -363.9 mm, Y = 559.8 mm, Z = 531.8 mm,       W = 0.4 deg, P = 0.5 deg,
    GP2:
        UF : 1, UT : 2,
       J1 = 0.0 deg, J2 = 0.0 deg
 };
P[234] {
    GP1:
        UF : 6, UT : 5,     CONFIG: 'N U T, 0, 0, 0',
       X = -381.1 mm, Y = 490.0 mm, Z = 531.8 mm,
       W = 0.4 deg, P = 0.4 deg,
    GP2:
        UF : 1, UT : 2,
       J1 = 0.0 deg, J2 = 0.0 deg
 };
P[504] {
    GP1:
        UF : 6, UT : 5,     CONFIG: 'N U T, 0, 0, 0',
 X = -364.1 mm, Y = 561.0 mm, Z = 531.8 mm,       W = 0.4 deg, P = 0.4 deg,
    GP2:
        UF : 1, UT : 2,
       J1 = 0.0 deg, J2 = 0.0 deg
 };
P[235] {
    GP1:
        UF : 6, UT : 5,     CONFIG: 'N U T, 0, 0, 0',
       X = -381.3 mm, Y = 491.4 mm, Z = 531.8 mm,
       W = 0.3 deg, P = 0.3 deg,
    GP2:
        UF : 1, UT : 2,
       J1 = 0.0 deg, J2 = 0.0 deg
 };
P[505] {
    GP1:
        UF : 6, UT : 5,     CONFIG: 'N U T, 0, 0, 0',
 X = -364.3 mm, Y = 562.4 mm, Z = 531.8 mm,       W = 0.3 deg, P = 0.3 deg,
    GP2:
        UF : 1, UT : 2,
       J1 = 0.0 deg, J2 = 0.0 deg
 };
P[236] {
    GP1:
        UF : 6, UT : 5,     CONFIG: 'N U T, 0, 0, 0',
       X = -381.8 mm, Y = 492.8 mm, Z = 531.8 mm,
       W = 0.3 deg, P = 0.3 deg,
    GP2:
        UF : 1, UT : 2,
       J1 = 0.0 deg, J2 = 0.0 deg
 };
P[506] {
    GP1:
        UF : 6, UT : 5,     CONFIG: 'N U T, 0, 0, 0',
 X = -364.8 mm, Y = 563.8 mm, Z = 531.8 mm,       W = 0.3 deg, P = 0.3 deg,
    GP2:
        UF : 1, UT : 2,
       J1 = 0.0 deg, J2 = 0.0 deg
 };
P[237] {
    GP1:
        UF : 6, UT : 5,     CONFIG: 'N U T, 0, 0, 0',
       X = -382.3 mm, Y = 493.8 mm, Z = 531.8 mm,
       W = 0.2 deg, P = 0.2 deg,
    GP2:
        UF : 1, UT : 2,
       J1 = 0.0 deg, J2 = 0.0 deg
 };
P[507] {
    GP1:
        UF : 6, UT : 5,     CONFIG: 'N U T, 0, 0, 0',
 X = -365.3 mm, Y = 564.8 mm, Z = 531.8 mm,       W = 0.2 deg, P = 0.2 deg,
    GP2:
        UF : 1, UT : 2,
       J1 = 0.0 deg, J2 = 0.0 deg
 };
P[238] {
    GP1:
        UF : 6, UT : 5,     CONFIG: 'N U T, 0, 0, 0',
       X = -383.0 mm, Y = 494.7 mm, Z = 531.8 mm,
       W = 0.2 deg, P = 0.2 deg,
    GP2:
        UF : 1, UT : 2,
       J1 = 0.0 deg, J2 = 0.0 deg
 };
P[508] {
    GP1:
        UF : 6, UT : 5,     CONFIG: 'N U T, 0, 0, 0',
 X = -366.0 mm, Y = 565.7 mm, Z = 531.8 mm,       W = 0.2 deg, P = 0.2 deg,
    GP2:
        UF : 1, UT : 2,
       J1 = 0.0 deg, J2 = 0.0 deg
 };
P[239] {
    GP1:
        UF : 6, UT : 5,     CONFIG: 'N U T, 0, 0, 0',
       X = -383.8 mm, Y = 495.7 mm, Z = 531.8 mm,
       W = 0.1 deg, P = 0.2 deg,
    GP2:
        UF : 1, UT : 2,
       J1 = 0.0 deg, J2 = 0.0 deg
 };
P[509] {
    GP1:
        UF : 6, UT : 5,     CONFIG: 'N U T, 0, 0, 0',
 X = -366.8 mm, Y = 566.7 mm, Z = 531.8 mm,       W = 0.1 deg, P = 0.2 deg,
    GP2:
        UF : 1, UT : 2,
       J1 = 0.0 deg, J2 = 0.0 deg
 };
P[240] {
    GP1:
        UF : 6, UT : 5,     CONFIG: 'N U T, 0, 0, 0',
       X = -385.5 mm, Y = 497.1 mm, Z = 531.8 mm,
       W = 0.1 deg, P = 0.1 deg,
    GP2:
        UF : 1, UT : 2,
       J1 = 0.0 deg, J2 = 0.0 deg
 };
P[510] {
    GP1:
        UF : 6, UT : 5,     CONFIG: 'N U T, 0, 0, 0',
 X = -368.5 mm, Y = 568.1 mm, Z = 531.8 mm,       W = 0.1 deg, P = 0.1 deg,
    GP2:
        UF : 1, UT : 2,
       J1 = 0.0 deg, J2 = 0.0 deg
 };
P[241] {
    GP1:
        UF : 6, UT : 5,     CONFIG: 'N U T, 0, 0, 0',
       X = -393.4 mm, Y = 502.4 mm, Z = 531.8 mm,
       W = 0.0 deg, P = 0.0 deg,
    GP2:
        UF : 1, UT : 2,
       J1 = 0.0 deg, J2 = 0.0 deg
 };
P[511] {
    GP1:
        UF : 6, UT : 5,     CONFIG: 'N U T, 0, 0, 0',
 X = -376.4 mm, Y = 573.4 mm, Z = 531.8 mm,       W = 0.0 deg, P = 0.0 deg,
    GP2:
        UF : 1, UT : 2,
       J1 = 0.0 deg, J2 = 0.0 deg
 };
P[242] {
    GP1:
        UF : 6, UT : 5,     CONFIG: 'N U T, 0, 0, 0',
       X = -401.5 mm, Y = 507.5 mm, Z = 531.8 mm,
       W = 0.0 deg, P = 0.0 deg,
    GP2:
        UF : 1, UT : 2,
       J1 = 0.0 deg, J2 = 0.0 deg
 };
P[512] {
    GP1:
        UF : 6, UT : 5,     CONFIG: 'N U T, 0, 0, 0',
 X = -384.5 mm, Y = 578.5 mm, Z = 531.8 mm,       W = 0.0 deg, P = 0.0 deg,
    GP2:
        UF : 1, UT : 2,
       J1 = 0.0 deg, J2 = 0.0 deg
 };
P[243] {
    GP1:
        UF : 6, UT : 5,     CONFIG: 'N U T, 0, 0, 0',
       X = -409.6 mm, Y = 512.5 mm, Z = 531.8 mm,
       W = 0.0 deg, P = 0.0 deg,
    GP2:
        UF : 1, UT : 2,
       J1 = 0.0 deg, J2 = 0.0 deg
 };
P[513] {
    GP1:
        UF : 6, UT : 5,     CONFIG: 'N U T, 0, 0, 0',
 X = -392.6 mm, Y = 583.5 mm, Z = 531.8 mm,       W = 0.0 deg, P = 0.0 deg,
    GP2:
        UF : 1, UT : 2,
       J1 = 0.0 deg, J2 = 0.0 deg
 };
P[244] {
    GP1:
        UF : 6, UT : 5,     CONFIG: 'N U T, 0, 0, 0',
       X = -417.9 mm, Y = 517.2 mm, Z = 531.8 mm,
       W = 0.0 deg, P = 0.0 deg,
    GP2:
        UF : 1, UT : 2,
       J1 = 0.0 deg, J2 = 0.0 deg
 };
P[514] {
    GP1:
        UF : 6, UT : 5,     CONFIG: 'N U T, 0, 0, 0',
 X = -400.9 mm, Y = 588.2 mm, Z = 531.8 mm,       W = 0.0 deg, P = 0.0 deg,
    GP2:
        UF : 1, UT : 2,
       J1 = 0.0 deg, J2 = 0.0 deg
 };
P[245] {
    GP1:
        UF : 6, UT : 5,     CONFIG: 'N U T, 0, 0, 0',
       X = -426.2 mm, Y = 521.9 mm, Z = 531.8 mm,
       W = 0.0 deg, P = 0.0 deg,
    GP2:
        UF : 1, UT : 2,
       J1 = 0.0 deg, J2 = 0.0 deg
 };
P[515] {
    GP1:
        UF : 6, UT : 5,     CONFIG: 'N U T, 0, 0, 0',
 X = -409.2 mm, Y = 592.9 mm, Z = 531.8 mm,       W = 0.0 deg, P = 0.0 deg,
    GP2:
        UF : 1, UT : 2,
       J1 = 0.0 deg, J2 = 0.0 deg
 };
P[246] {
    GP1:
        UF : 6, UT : 5,     CONFIG: 'N U T, 0, 0, 0',
       X = -434.6 mm, Y = 526.3 mm, Z = 531.8 mm,
       W = 0.0 deg, P = 0.0 deg,
    GP2:
        UF : 1, UT : 2,
       J1 = 0.0 deg, J2 = 0.0 deg
 };
P[516] {
    GP1:
        UF : 6, UT : 5,     CONFIG: 'N U T, 0, 0, 0',
 X = -417.6 mm, Y = 597.3 mm, Z = 531.8 mm,       W = 0.0 deg, P = 0.0 deg,
    GP2:
        UF : 1, UT : 2,
       J1 = 0.0 deg, J2 = 0.0 deg
 };
P[247] {
    GP1:
        UF : 6, UT : 5,     CONFIG: 'N U T, 0, 0, 0',
       X = -441.0 mm, Y = 529.7 mm, Z = 531.8 mm,
       W = 0.0 deg, P = 0.0 deg,
    GP2:
        UF : 1, UT : 2,
       J1 = 0.0 deg, J2 = 0.0 deg
 };
P[517] {
    GP1:
        UF : 6, UT : 5,     CONFIG: 'N U T, 0, 0, 0',
 X = -424.0 mm, Y = 600.7 mm, Z = 531.8 mm,       W = 0.0 deg, P = 0.0 deg,
    GP2:
        UF : 1, UT : 2,
       J1 = 0.0 deg, J2 = 0.0 deg
 };
P[248] {
    GP1:
        UF : 6, UT : 5,     CONFIG: 'N U T, 0, 0, 0',
       X = -443.4 mm, Y = 531.2 mm, Z = 531.8 mm,
       W = 0.0 deg, P = 0.0 deg,
    GP2:
        UF : 1, UT : 2,
       J1 = 0.0 deg, J2 = 0.0 deg
 };
P[518] {
    GP1:
        UF : 6, UT : 5,     CONFIG: 'N U T, 0, 0, 0',
 X = -426.4 mm, Y = 602.2 mm, Z = 531.8 mm,       W = 0.0 deg, P = 0.0 deg,
    GP2:
        UF : 1, UT : 2,
       J1 = 0.0 deg, J2 = 0.0 deg
 };
P[249] {
    GP1:
        UF : 6, UT : 5,     CONFIG: 'N U T, 0, 0, 0',
       X = -445.5 mm, Y = 533.1 mm, Z = 531.8 mm,
       W = 0.0 deg, P = 0.0 deg,
    GP2:
        UF : 1, UT : 2,
       J1 = 0.0 deg, J2 = 0.0 deg
 };
P[519] {
    GP1:
        UF : 6, UT : 5,     CONFIG: 'N U T, 0, 0, 0',
 X = -428.5 mm, Y = 604.1 mm, Z = 531.8 mm,       W = 0.0 deg, P = 0.0 deg,
    GP2:
        UF : 1, UT : 2,
       J1 = 0.0 deg, J2 = 0.0 deg
 };
P[250] {
    GP1:
        UF : 6, UT : 5,     CONFIG: 'N U T, 0, 0, 0',
       X = -447.2 mm, Y = 535.3 mm, Z = 531.8 mm,
       W = 0.0 deg, P = 0.0 deg,
    GP2:
        UF : 1, UT : 2,
       J1 = 0.0 deg, J2 = 0.0 deg
 };
P[520] {
    GP1:
        UF : 6, UT : 5,     CONFIG: 'N U T, 0, 0, 0',
 X = -430.2 mm, Y = 606.3 mm, Z = 531.8 mm,       W = 0.0 deg, P = 0.0 deg,
    GP2:
        UF : 1, UT : 2,
       J1 = 0.0 deg, J2 = 0.0 deg
 };
P[251] {
    GP1:
        UF : 6, UT : 5,     CONFIG: 'N U T, 0, 0, 0',
       X = -452.3 mm, Y = 543.6 mm, Z = 531.8 mm,
       W = 0.0 deg, P = 0.0 deg,
    GP2:
        UF : 1, UT : 2,
       J1 = 0.0 deg, J2 = 0.0 deg
 };
P[521] {
    GP1:
        UF : 6, UT : 5,     CONFIG: 'N U T, 0, 0, 0',
 X = -435.3 mm, Y = 614.6 mm, Z = 531.8 mm,       W = 0.0 deg, P = 0.0 deg,
    GP2:
        UF : 1, UT : 2,
       J1 = 0.0 deg, J2 = 0.0 deg
 };
P[252] {
    GP1:
        UF : 6, UT : 5,     CONFIG: 'N U T, 0, 0, 0',
       X = -457.3 mm, Y = 552.1 mm, Z = 531.8 mm,
       W = 0.0 deg, P = 0.0 deg,
    GP2:
        UF : 1, UT : 2,
       J1 = 0.0 deg, J2 = 0.0 deg
 };
P[522] {
    GP1:
        UF : 6, UT : 5,     CONFIG: 'N U T, 0, 0, 0',
 X = -440.3 mm, Y = 623.1 mm, Z = 531.8 mm,       W = 0.0 deg, P = 0.0 deg,
    GP2:
        UF : 1, UT : 2,
       J1 = 0.0 deg, J2 = 0.0 deg
 };
P[253] {
    GP1:
        UF : 6, UT : 5,     CONFIG: 'N U T, 0, 0, 0',
       X = -457.8 mm, Y = 553.3 mm, Z = 531.8 mm,
       W = 0.0 deg, P = 0.0 deg,
    GP2:
        UF : 1, UT : 2,
       J1 = 0.0 deg, J2 = 0.0 deg
 };
P[523] {
    GP1:
        UF : 6, UT : 5,     CONFIG: 'N U T, 0, 0, 0',
 X = -440.8 mm, Y = 624.3 mm, Z = 531.8 mm,       W = 0.0 deg, P = 0.0 deg,
    GP2:
        UF : 1, UT : 2,
       J1 = 0.0 deg, J2 = 0.0 deg
 };
P[254] {
    GP1:
        UF : 6, UT : 5,     CONFIG: 'N U T, 0, 0, 0',
       X = -458.2 mm, Y = 554.9 mm, Z = 531.8 mm,
       W = 0.0 deg, P = 0.0 deg,
    GP2:
        UF : 1, UT : 2,
       J1 = 0.0 deg, J2 = 0.0 deg
 };
P[524] {
    GP1:
        UF : 6, UT : 5,     CONFIG: 'N U T, 0, 0, 0',
 X = -441.2 mm, Y = 625.9 mm, Z = 531.8 mm,       W = 0.0 deg, P = 0.0 deg,
    GP2:
        UF : 1, UT : 2,
       J1 = 0.0 deg, J2 = 0.0 deg
 };
P[255] {
    GP1:
        UF : 6, UT : 5,     CONFIG: 'N U T, 0, 0, 0',
       X = -458.2 mm, Y = 557.0 mm, Z = 531.8 mm,
       W = 0.0 deg, P = 0.0 deg,
    GP2:
        UF : 1, UT : 2,
       J1 = 0.0 deg, J2 = 0.0 deg
 };
P[525] {
    GP1:
        UF : 6, UT : 5,     CONFIG: 'N U T, 0, 0, 0',
 X = -441.2 mm, Y = 628.0 mm, Z = 531.8 mm,       W = 0.0 deg, P = 0.0 deg,
    GP2:
        UF : 1, UT : 2,
       J1 = 0.0 deg, J2 = 0.0 deg
 };
P[256] {
    GP1:
        UF : 6, UT : 5,     CONFIG: 'N U T, 0, 0, 0',
       X = -457.9 mm, Y = 558.6 mm, Z = 531.8 mm,
       W = 0.0 deg, P = 0.0 deg,
    GP2:
        UF : 1, UT : 2,
       J1 = 0.0 deg, J2 = 0.0 deg
 };
P[526] {
    GP1:
        UF : 6, UT : 5,     CONFIG: 'N U T, 0, 0, 0',
 X = -440.9 mm, Y = 629.6 mm, Z = 531.8 mm,       W = 0.0 deg, P = 0.0 deg,
    GP2:
        UF : 1, UT : 2,
       J1 = 0.0 deg, J2 = 0.0 deg
 };
P[257] {
    GP1:
        UF : 6, UT : 5,     CONFIG: 'N U T, 0, 0, 0',
       X = -457.2 mm, Y = 560.0 mm, Z = 531.8 mm,
       W = 0.0 deg, P = 0.0 deg,
    GP2:
        UF : 1, UT : 2,
       J1 = 0.0 deg, J2 = 0.0 deg
 };
P[527] {
    GP1:
        UF : 6, UT : 5,     CONFIG: 'N U T, 0, 0, 0',
 X = -440.2 mm, Y = 631.0 mm, Z = 531.8 mm,       W = 0.0 deg, P = 0.0 deg,
    GP2:
        UF : 1, UT : 2,
       J1 = 0.0 deg, J2 = 0.0 deg
 };
P[258] {
    GP1:
        UF : 6, UT : 5,     CONFIG: 'N U T, 0, 0, 0',
       X = -456.2 mm, Y = 561.4 mm, Z = 531.8 mm,
       W = 0.0 deg, P = 0.0 deg,
    GP2:
        UF : 1, UT : 2,
       J1 = 0.0 deg, J2 = 0.0 deg
 };
P[528] {
    GP1:
        UF : 6, UT : 5,     CONFIG: 'N U T, 0, 0, 0',
 X = -439.2 mm, Y = 632.4 mm, Z = 531.8 mm,       W = 0.0 deg, P = 0.0 deg,
    GP2:
        UF : 1, UT : 2,
       J1 = 0.0 deg, J2 = 0.0 deg
 };
P[259] {
    GP1:
        UF : 6, UT : 5,     CONFIG: 'N U T, 0, 0, 0',
       X = -455.1 mm, Y = 562.4 mm, Z = 531.8 mm,
       W = 0.0 deg, P = 0.0 deg,
    GP2:
        UF : 1, UT : 2,
       J1 = 0.0 deg, J2 = 0.0 deg
 };
P[529] {
    GP1:
        UF : 6, UT : 5,     CONFIG: 'N U T, 0, 0, 0',
 X = -438.1 mm, Y = 633.4 mm, Z = 531.8 mm,       W = 0.0 deg, P = 0.0 deg,
    GP2:
        UF : 1, UT : 2,
       J1 = 0.0 deg, J2 = 0.0 deg
 };
P[260] {
    GP1:
        UF : 6, UT : 5,     CONFIG: 'N U T, 0, 0, 0',
       X = -447.0 mm, Y = 567.7 mm, Z = 531.8 mm,
       W = 0.0 deg, P = 0.0 deg,
    GP2:
        UF : 1, UT : 2,
       J1 = 0.0 deg, J2 = 0.0 deg
 };
P[530] {
    GP1:
        UF : 6, UT : 5,     CONFIG: 'N U T, 0, 0, 0',
 X = -430.0 mm, Y = 638.7 mm, Z = 531.8 mm,       W = 0.0 deg, P = 0.0 deg,
    GP2:
        UF : 1, UT : 2,
       J1 = 0.0 deg, J2 = 0.0 deg
 };
P[261] {
    GP1:
        UF : 6, UT : 5,     CONFIG: 'N U T, 0, 0, 0',
       X = -439.0 mm, Y = 572.9 mm, Z = 531.8 mm,
       W = 0.0 deg, P = 0.0 deg,
    GP2:
        UF : 1, UT : 2,
       J1 = 0.0 deg, J2 = 0.0 deg
 };
P[531] {
    GP1:
        UF : 6, UT : 5,     CONFIG: 'N U T, 0, 0, 0',
 X = -422.0 mm, Y = 643.9 mm, Z = 531.8 mm,       W = 0.0 deg, P = 0.0 deg,
    GP2:
        UF : 1, UT : 2,
       J1 = 0.0 deg, J2 = 0.0 deg
 };
P[262] {
    GP1:
        UF : 6, UT : 5,     CONFIG: 'N U T, 0, 0, 0',
       X = -430.9 mm, Y = 578.1 mm, Z = 531.8 mm,
       W = 0.0 deg, P = 0.0 deg,
    GP2:
        UF : 1, UT : 2,
       J1 = 0.0 deg, J2 = 0.0 deg
 };
P[532] {
    GP1:
        UF : 6, UT : 5,     CONFIG: 'N U T, 0, 0, 0',
 X = -413.9 mm, Y = 649.1 mm, Z = 531.8 mm,       W = 0.0 deg, P = 0.0 deg,
    GP2:
        UF : 1, UT : 2,
       J1 = 0.0 deg, J2 = 0.0 deg
 };
P[263] {
    GP1:
        UF : 6, UT : 5,     CONFIG: 'N U T, 0, 0, 0',
       X = -422.8 mm, Y = 583.4 mm, Z = 531.8 mm,
       W = 0.0 deg, P = 0.0 deg,
    GP2:
        UF : 1, UT : 2,
       J1 = 0.0 deg, J2 = 0.0 deg
 };
P[533] {
    GP1:
        UF : 6, UT : 5,     CONFIG: 'N U T, 0, 0, 0',
 X = -405.8 mm, Y = 654.4 mm, Z = 531.8 mm,       W = 0.0 deg, P = 0.0 deg,
    GP2:
        UF : 1, UT : 2,
       J1 = 0.0 deg, J2 = 0.0 deg
 };
P[264] {
    GP1:
        UF : 6, UT : 5,     CONFIG: 'N U T, 0, 0, 0',
       X = -414.7 mm, Y = 588.6 mm, Z = 531.8 mm,
       W = 0.0 deg, P = 0.0 deg,
    GP2:
        UF : 1, UT : 2,
       J1 = 0.0 deg, J2 = 0.0 deg
 };
P[534] {
    GP1:
        UF : 6, UT : 5,     CONFIG: 'N U T, 0, 0, 0',
 X = -397.7 mm, Y = 659.6 mm, Z = 531.8 mm,       W = 0.0 deg, P = 0.0 deg,
    GP2:
        UF : 1, UT : 2,
       J1 = 0.0 deg, J2 = 0.0 deg
 };
P[265] {
    GP1:
        UF : 6, UT : 5,     CONFIG: 'N U T, 0, 0, 0',
       X = -406.7 mm, Y = 593.9 mm, Z = 531.8 mm,
       W = 0.0 deg, P = 0.0 deg,
    GP2:
        UF : 1, UT : 2,
       J1 = 0.0 deg, J2 = 0.0 deg
 };
P[535] {
    GP1:
        UF : 6, UT : 5,     CONFIG: 'N U T, 0, 0, 0',
 X = -389.7 mm, Y = 664.9 mm, Z = 531.8 mm,       W = 0.0 deg, P = 0.0 deg,
    GP2:
        UF : 1, UT : 2,
       J1 = 0.0 deg, J2 = 0.0 deg
 };
P[266] {
    GP1:
        UF : 6, UT : 5,     CONFIG: 'N U T, 0, 0, 0',
       X = -398.6 mm, Y = 599.1 mm, Z = 531.8 mm,
       W = 0.0 deg, P = 0.0 deg,
    GP2:
        UF : 1, UT : 2,
       J1 = 0.0 deg, J2 = 0.0 deg
 };
P[536] {
    GP1:
        UF : 6, UT : 5,     CONFIG: 'N U T, 0, 0, 0',
 X = -381.6 mm, Y = 670.1 mm, Z = 531.8 mm,       W = 0.0 deg, P = 0.0 deg,
    GP2:
        UF : 1, UT : 2,
       J1 = 0.0 deg, J2 = 0.0 deg
 };
P[267] {
    GP1:
        UF : 6, UT : 5,     CONFIG: 'N U T, 0, 0, 0',
       X = -390.5 mm, Y = 604.4 mm, Z = 531.8 mm,
       W = 0.0 deg, P = 0.0 deg,
    GP2:
        UF : 1, UT : 2,
       J1 = 0.0 deg, J2 = 0.0 deg
 };
P[537] {
    GP1:
        UF : 6, UT : 5,     CONFIG: 'N U T, 0, 0, 0',
 X = -373.5 mm, Y = 675.4 mm, Z = 531.8 mm,       W = 0.0 deg, P = 0.0 deg,
    GP2:
        UF : 1, UT : 2,
       J1 = 0.0 deg, J2 = 0.0 deg
 };
P[268] {
    GP1:
        UF : 6, UT : 5,     CONFIG: 'N U T, 0, 0, 0',
       X = -382.5 mm, Y = 609.6 mm, Z = 531.8 mm,
       W = 0.0 deg, P = 0.0 deg,
    GP2:
        UF : 1, UT : 2,
       J1 = 0.0 deg, J2 = 0.0 deg
 };
P[538] {
    GP1:
        UF : 6, UT : 5,     CONFIG: 'N U T, 0, 0, 0',
 X = -365.5 mm, Y = 680.6 mm, Z = 531.8 mm,       W = 0.0 deg, P = 0.0 deg,
    GP2:
        UF : 1, UT : 2,
       J1 = 0.0 deg, J2 = 0.0 deg
 };
/END
